SUBAPPLICATION InputOutputTesterButton_AI_Calibrate_3P_OPC_UA (* AI Calibrate 3P Tester (OPC-UA): 8 Analog-Eingaenge mit 3-Punkt-Kalibrierung (Rohwert+kalibrierter Wert+Bargraph+C_MIN/C_MID/C_MAX, fuer Sensoren mit Mittelstellung) + 12 unveraenderte digitale Ausgaenge *)
  (* Standard: 61499-2; Description: Copyright (c) 2026 Meisterschulen am Ostbahnhof This program and the accompanying materials are made available under the terms of the Eclipse Public License 2.0 which is available at https://www.eclipse.org/legal/epl-2.0/ SPDX-License-Identifier: EPL-2.0 *)
  (* Version 1.0, 2026-09-11, Franz Höpfinger, Meisterschulen am Ostbahnhof, 3-Punkt-Pendant zu InputOutputTesterButton_AI_Calibrate_OPC_UA - logiBUS_AI_Calibrate_3P_IDA_OPC statt logiBUS_AI_Calibrate_IDA_OPC (C_MIN/C_MID/C_MAX statt CO/CS) *)
  (* Version 1.1, 2026-09-20, Franz Höpfinger, Meisterschulen am Ostbahnhof, Rohwert-Anzeige an den 3 Kalibrierpunkten (Min/Mid/Max-Raw) fuer alle 8 Kanaele ergaenzt, siehe logiBUS_AI_Calibrate_3P_IDA_OPC v1.8. Neue Parameter stObjMinRaw/stObjMidRaw/stObjMaxRaw + ID_MIN/MID/MAX_RAW_WRITE pro Kanal, neue VT-Objekte NumberVariable_AIC_I0N_MINRAW/_MIDRAW/_MAXRAW_N (DefaultPool_AIC_3P_Numeric, IDs 21040-21063) + OPC-UA-Adressen AIC_I0N_MIN/MID/MAX_RAW_WRITE (SubStrings). *)
  PACKAGE Meins::InputOutputTester::Button_AI_Calibrate_3P_OPC_UA;
  IMPORT Meins::InputOutputTester::Button_AI_Calibrate_3P_OPC_UA::SubStrings::AIC_I1_RAW_WRITE;
  IMPORT Meins::InputOutputTester::Button_AI_Calibrate_3P_OPC_UA::SubStrings::AIC_I1_CAL_WRITE;
  IMPORT Meins::InputOutputTester::Button_AI_Calibrate_3P_OPC_UA::SubStrings::AIC_I2_RAW_WRITE;
  IMPORT Meins::InputOutputTester::Button_AI_Calibrate_3P_OPC_UA::SubStrings::AIC_I2_CAL_WRITE;
  IMPORT Meins::InputOutputTester::Button_AI_Calibrate_3P_OPC_UA::SubStrings::AIC_I3_RAW_WRITE;
  IMPORT Meins::InputOutputTester::Button_AI_Calibrate_3P_OPC_UA::SubStrings::AIC_I3_CAL_WRITE;
  IMPORT Meins::InputOutputTester::Button_AI_Calibrate_3P_OPC_UA::SubStrings::AIC_I4_RAW_WRITE;
  IMPORT Meins::InputOutputTester::Button_AI_Calibrate_3P_OPC_UA::SubStrings::AIC_I4_CAL_WRITE;
  IMPORT Meins::InputOutputTester::Button_AI_Calibrate_3P_OPC_UA::SubStrings::AIC_I5_RAW_WRITE;
  IMPORT Meins::InputOutputTester::Button_AI_Calibrate_3P_OPC_UA::SubStrings::AIC_I5_CAL_WRITE;
  IMPORT Meins::InputOutputTester::Button_AI_Calibrate_3P_OPC_UA::SubStrings::AIC_I6_RAW_WRITE;
  IMPORT Meins::InputOutputTester::Button_AI_Calibrate_3P_OPC_UA::SubStrings::AIC_I6_CAL_WRITE;
  IMPORT Meins::InputOutputTester::Button_AI_Calibrate_3P_OPC_UA::SubStrings::AIC_I7_RAW_WRITE;
  IMPORT Meins::InputOutputTester::Button_AI_Calibrate_3P_OPC_UA::SubStrings::AIC_I7_CAL_WRITE;
  IMPORT Meins::InputOutputTester::Button_AI_Calibrate_3P_OPC_UA::SubStrings::AIC_I8_RAW_WRITE;
  IMPORT Meins::InputOutputTester::Button_AI_Calibrate_3P_OPC_UA::SubStrings::AIC_I8_CAL_WRITE;
  IMPORT Meins::InputOutputTester::Button_AI_Calibrate_3P_OPC_UA::SubStrings::AIC_I1_MIN_METHOD;
  IMPORT Meins::InputOutputTester::Button_AI_Calibrate_3P_OPC_UA::SubStrings::AIC_I1_MID_METHOD;
  IMPORT Meins::InputOutputTester::Button_AI_Calibrate_3P_OPC_UA::SubStrings::AIC_I1_MAX_METHOD;
  IMPORT Meins::InputOutputTester::Button_AI_Calibrate_3P_OPC_UA::SubStrings::AIC_I2_MIN_METHOD;
  IMPORT Meins::InputOutputTester::Button_AI_Calibrate_3P_OPC_UA::SubStrings::AIC_I2_MID_METHOD;
  IMPORT Meins::InputOutputTester::Button_AI_Calibrate_3P_OPC_UA::SubStrings::AIC_I2_MAX_METHOD;
  IMPORT Meins::InputOutputTester::Button_AI_Calibrate_3P_OPC_UA::SubStrings::AIC_I3_MIN_METHOD;
  IMPORT Meins::InputOutputTester::Button_AI_Calibrate_3P_OPC_UA::SubStrings::AIC_I3_MID_METHOD;
  IMPORT Meins::InputOutputTester::Button_AI_Calibrate_3P_OPC_UA::SubStrings::AIC_I3_MAX_METHOD;
  IMPORT Meins::InputOutputTester::Button_AI_Calibrate_3P_OPC_UA::SubStrings::AIC_I4_MIN_METHOD;
  IMPORT Meins::InputOutputTester::Button_AI_Calibrate_3P_OPC_UA::SubStrings::AIC_I4_MID_METHOD;
  IMPORT Meins::InputOutputTester::Button_AI_Calibrate_3P_OPC_UA::SubStrings::AIC_I4_MAX_METHOD;
  IMPORT Meins::InputOutputTester::Button_AI_Calibrate_3P_OPC_UA::SubStrings::AIC_I5_MIN_METHOD;
  IMPORT Meins::InputOutputTester::Button_AI_Calibrate_3P_OPC_UA::SubStrings::AIC_I5_MID_METHOD;
  IMPORT Meins::InputOutputTester::Button_AI_Calibrate_3P_OPC_UA::SubStrings::AIC_I5_MAX_METHOD;
  IMPORT Meins::InputOutputTester::Button_AI_Calibrate_3P_OPC_UA::SubStrings::AIC_I6_MIN_METHOD;
  IMPORT Meins::InputOutputTester::Button_AI_Calibrate_3P_OPC_UA::SubStrings::AIC_I6_MID_METHOD;
  IMPORT Meins::InputOutputTester::Button_AI_Calibrate_3P_OPC_UA::SubStrings::AIC_I6_MAX_METHOD;
  IMPORT Meins::InputOutputTester::Button_AI_Calibrate_3P_OPC_UA::SubStrings::AIC_I7_MIN_METHOD;
  IMPORT Meins::InputOutputTester::Button_AI_Calibrate_3P_OPC_UA::SubStrings::AIC_I7_MID_METHOD;
  IMPORT Meins::InputOutputTester::Button_AI_Calibrate_3P_OPC_UA::SubStrings::AIC_I7_MAX_METHOD;
  IMPORT Meins::InputOutputTester::Button_AI_Calibrate_3P_OPC_UA::SubStrings::AIC_I8_MIN_METHOD;
  IMPORT Meins::InputOutputTester::Button_AI_Calibrate_3P_OPC_UA::SubStrings::AIC_I8_MID_METHOD;
  IMPORT Meins::InputOutputTester::Button_AI_Calibrate_3P_OPC_UA::SubStrings::AIC_I8_MAX_METHOD;
  IMPORT Meins::InputOutputTester::Button_AI_Calibrate_3P_OPC_UA::SubStrings::Q01_READ;
  IMPORT Meins::InputOutputTester::Button_AI_Calibrate_3P_OPC_UA::SubStrings::Q01_WRITE;
  IMPORT Meins::InputOutputTester::Button_AI_Calibrate_3P_OPC_UA::SubStrings::Q02_READ;
  IMPORT Meins::InputOutputTester::Button_AI_Calibrate_3P_OPC_UA::SubStrings::Q02_WRITE;
  IMPORT Meins::InputOutputTester::Button_AI_Calibrate_3P_OPC_UA::SubStrings::Q03_READ;
  IMPORT Meins::InputOutputTester::Button_AI_Calibrate_3P_OPC_UA::SubStrings::Q03_WRITE;
  IMPORT Meins::InputOutputTester::Button_AI_Calibrate_3P_OPC_UA::SubStrings::Q04_READ;
  IMPORT Meins::InputOutputTester::Button_AI_Calibrate_3P_OPC_UA::SubStrings::Q04_WRITE;
  IMPORT Meins::InputOutputTester::Button_AI_Calibrate_3P_OPC_UA::SubStrings::Q05_READ;
  IMPORT Meins::InputOutputTester::Button_AI_Calibrate_3P_OPC_UA::SubStrings::Q05_WRITE;
  IMPORT Meins::InputOutputTester::Button_AI_Calibrate_3P_OPC_UA::SubStrings::Q06_READ;
  IMPORT Meins::InputOutputTester::Button_AI_Calibrate_3P_OPC_UA::SubStrings::Q06_WRITE;
  IMPORT Meins::InputOutputTester::Button_AI_Calibrate_3P_OPC_UA::SubStrings::Q07_READ;
  IMPORT Meins::InputOutputTester::Button_AI_Calibrate_3P_OPC_UA::SubStrings::Q07_WRITE;
  IMPORT Meins::InputOutputTester::Button_AI_Calibrate_3P_OPC_UA::SubStrings::Q08_READ;
  IMPORT Meins::InputOutputTester::Button_AI_Calibrate_3P_OPC_UA::SubStrings::Q08_WRITE;
  IMPORT Meins::InputOutputTester::Button_AI_Calibrate_3P_OPC_UA::SubStrings::Q09_READ;
  IMPORT Meins::InputOutputTester::Button_AI_Calibrate_3P_OPC_UA::SubStrings::Q09_WRITE;
  IMPORT Meins::InputOutputTester::Button_AI_Calibrate_3P_OPC_UA::SubStrings::Q10_READ;
  IMPORT Meins::InputOutputTester::Button_AI_Calibrate_3P_OPC_UA::SubStrings::Q10_WRITE;
  IMPORT Meins::InputOutputTester::Button_AI_Calibrate_3P_OPC_UA::SubStrings::Q11_READ;
  IMPORT Meins::InputOutputTester::Button_AI_Calibrate_3P_OPC_UA::SubStrings::Q11_WRITE;
  IMPORT Meins::InputOutputTester::Button_AI_Calibrate_3P_OPC_UA::SubStrings::Q12_READ;
  IMPORT Meins::InputOutputTester::Button_AI_Calibrate_3P_OPC_UA::SubStrings::Q12_WRITE;
  IMPORT Meins::InputOutputTester::Button_AI_Calibrate_3P_OPC_UA::SubStrings::Tick_WRITE;
  IMPORT Uebungen::const::UT::AIC::DefaultPool_AIC_2P::NumberVariable_AIC_RAW_I01;
  IMPORT Uebungen::const::UT::AIC::DefaultPool_AIC_2P::NumberVariable_AIC_RAW_I02;
  IMPORT Uebungen::const::UT::AIC::DefaultPool_AIC_2P::NumberVariable_AIC_RAW_I03;
  IMPORT Uebungen::const::UT::AIC::DefaultPool_AIC_2P::NumberVariable_AIC_RAW_I04;
  IMPORT Uebungen::const::UT::AIC::DefaultPool_AIC_2P::NumberVariable_AIC_RAW_I05;
  IMPORT Uebungen::const::UT::AIC::DefaultPool_AIC_2P::NumberVariable_AIC_RAW_I06;
  IMPORT Uebungen::const::UT::AIC::DefaultPool_AIC_2P::NumberVariable_AIC_RAW_I07;
  IMPORT Uebungen::const::UT::AIC::DefaultPool_AIC_2P::NumberVariable_AIC_RAW_I08;
  IMPORT Uebungen::const::UT::AIC::DefaultPool_AIC_3P_Numeric::NumberVariable_AIC_CAL_I01_N;
  IMPORT Uebungen::const::UT::AIC::DefaultPool_AIC_3P_Numeric::NumberVariable_AIC_CAL_I02_N;
  IMPORT Uebungen::const::UT::AIC::DefaultPool_AIC_3P_Numeric::NumberVariable_AIC_CAL_I03_N;
  IMPORT Uebungen::const::UT::AIC::DefaultPool_AIC_3P_Numeric::NumberVariable_AIC_CAL_I04_N;
  IMPORT Uebungen::const::UT::AIC::DefaultPool_AIC_3P_Numeric::NumberVariable_AIC_CAL_I05_N;
  IMPORT Uebungen::const::UT::AIC::DefaultPool_AIC_3P_Numeric::NumberVariable_AIC_CAL_I06_N;
  IMPORT Uebungen::const::UT::AIC::DefaultPool_AIC_3P_Numeric::NumberVariable_AIC_CAL_I07_N;
  IMPORT Uebungen::const::UT::AIC::DefaultPool_AIC_3P_Numeric::NumberVariable_AIC_CAL_I08_N;
  IMPORT Uebungen::const::UT::AIC::DefaultPool_AIC_3P::Button_AIC_I01_CO;
  IMPORT Uebungen::const::UT::AIC::DefaultPool_AIC_3P::Button_AIC_I01_MID;
  IMPORT Uebungen::const::UT::AIC::DefaultPool_AIC_3P::Button_AIC_I01_CS;
  IMPORT Uebungen::const::UT::AIC::DefaultPool_AIC_3P::Button_AIC_I02_CO;
  IMPORT Uebungen::const::UT::AIC::DefaultPool_AIC_3P::Button_AIC_I02_MID;
  IMPORT Uebungen::const::UT::AIC::DefaultPool_AIC_3P::Button_AIC_I02_CS;
  IMPORT Uebungen::const::UT::AIC::DefaultPool_AIC_3P::Button_AIC_I03_CO;
  IMPORT Uebungen::const::UT::AIC::DefaultPool_AIC_3P::Button_AIC_I03_MID;
  IMPORT Uebungen::const::UT::AIC::DefaultPool_AIC_3P::Button_AIC_I03_CS;
  IMPORT Uebungen::const::UT::AIC::DefaultPool_AIC_3P::Button_AIC_I04_CO;
  IMPORT Uebungen::const::UT::AIC::DefaultPool_AIC_3P::Button_AIC_I04_MID;
  IMPORT Uebungen::const::UT::AIC::DefaultPool_AIC_3P::Button_AIC_I04_CS;
  IMPORT Uebungen::const::UT::AIC::DefaultPool_AIC_3P::Button_AIC_I05_CO;
  IMPORT Uebungen::const::UT::AIC::DefaultPool_AIC_3P::Button_AIC_I05_MID;
  IMPORT Uebungen::const::UT::AIC::DefaultPool_AIC_3P::Button_AIC_I05_CS;
  IMPORT Uebungen::const::UT::AIC::DefaultPool_AIC_3P::Button_AIC_I06_CO;
  IMPORT Uebungen::const::UT::AIC::DefaultPool_AIC_3P::Button_AIC_I06_MID;
  IMPORT Uebungen::const::UT::AIC::DefaultPool_AIC_3P::Button_AIC_I06_CS;
  IMPORT Uebungen::const::UT::AIC::DefaultPool_AIC_3P::Button_AIC_I07_CO;
  IMPORT Uebungen::const::UT::AIC::DefaultPool_AIC_3P::Button_AIC_I07_MID;
  IMPORT Uebungen::const::UT::AIC::DefaultPool_AIC_3P::Button_AIC_I07_CS;
  IMPORT Uebungen::const::UT::AIC::DefaultPool_AIC_3P::Button_AIC_I08_CO;
  IMPORT Uebungen::const::UT::AIC::DefaultPool_AIC_3P::Button_AIC_I08_MID;
  IMPORT Uebungen::const::UT::AIC::DefaultPool_AIC_3P::Button_AIC_I08_CS;
  IMPORT Uebungen::const::UT::AIC::DefaultPool_AIC_2P::Button_Q01;
  IMPORT Uebungen::const::UT::AIC::DefaultPool_AIC_2P::Button_Q02;
  IMPORT Uebungen::const::UT::AIC::DefaultPool_AIC_2P::Button_Q03;
  IMPORT Uebungen::const::UT::AIC::DefaultPool_AIC_2P::Button_Q04;
  IMPORT Uebungen::const::UT::AIC::DefaultPool_AIC_2P::Button_Q05;
  IMPORT Uebungen::const::UT::AIC::DefaultPool_AIC_2P::Button_Q06;
  IMPORT Uebungen::const::UT::AIC::DefaultPool_AIC_2P::Button_Q07;
  IMPORT Uebungen::const::UT::AIC::DefaultPool_AIC_2P::Button_Q08;
  IMPORT Uebungen::const::UT::AIC::DefaultPool_AIC_2P::Button_Q09;
  IMPORT Uebungen::const::UT::AIC::DefaultPool_AIC_2P::Button_Q10;
  IMPORT Uebungen::const::UT::AIC::DefaultPool_AIC_2P::Button_Q11;
  IMPORT Uebungen::const::UT::AIC::DefaultPool_AIC_2P::Button_Q12;
  IMPORT Uebungen::const::UT::AIC::DefaultPool_AIC_2P::OutputNumber_Tick;
  IMPORT logiBUS::io::AI::logiBUS_AI::AnalogInput_I1;
  IMPORT logiBUS::io::AI::logiBUS_AI::AnalogInput_I2;
  IMPORT logiBUS::io::AI::logiBUS_AI::AnalogInput_I3;
  IMPORT logiBUS::io::AI::logiBUS_AI::AnalogInput_I4;
  IMPORT logiBUS::io::AI::logiBUS_AI::AnalogInput_I5;
  IMPORT logiBUS::io::AI::logiBUS_AI::AnalogInput_I6;
  IMPORT logiBUS::io::AI::logiBUS_AI::AnalogInput_I7;
  IMPORT logiBUS::io::AI::logiBUS_AI::AnalogInput_I8;
  IMPORT logiBUS::io::DQ::logiBUS_DO::Output_Q1;
  IMPORT logiBUS::io::DQ::logiBUS_DO::Output_Q10;
  IMPORT logiBUS::io::DQ::logiBUS_DO::Output_Q11;
  IMPORT logiBUS::io::DQ::logiBUS_DO::Output_Q12;
  IMPORT logiBUS::io::DQ::logiBUS_DO::Output_Q2;
  IMPORT logiBUS::io::DQ::logiBUS_DO::Output_Q3;
  IMPORT logiBUS::io::DQ::logiBUS_DO::Output_Q4;
  IMPORT logiBUS::io::DQ::logiBUS_DO::Output_Q5;
  IMPORT logiBUS::io::DQ::logiBUS_DO::Output_Q6;
  IMPORT logiBUS::io::DQ::logiBUS_DO::Output_Q7;
  IMPORT logiBUS::io::DQ::logiBUS_DO::Output_Q8;
  IMPORT logiBUS::io::DQ::logiBUS_DO::Output_Q9;
  IMPORT Meins::InputOutputTester::Button_AI_Calibrate_3P_OPC_UA::SubStrings::AIC_I1_MINREF_READ;
  IMPORT Meins::InputOutputTester::Button_AI_Calibrate_3P_OPC_UA::SubStrings::AIC_I1_MINREF_WRITE;
  IMPORT Meins::InputOutputTester::Button_AI_Calibrate_3P_OPC_UA::SubStrings::AIC_I1_MIDREF_READ;
  IMPORT Meins::InputOutputTester::Button_AI_Calibrate_3P_OPC_UA::SubStrings::AIC_I1_MIDREF_WRITE;
  IMPORT Meins::InputOutputTester::Button_AI_Calibrate_3P_OPC_UA::SubStrings::AIC_I1_MAXREF_READ;
  IMPORT Meins::InputOutputTester::Button_AI_Calibrate_3P_OPC_UA::SubStrings::AIC_I1_MAXREF_WRITE;
  IMPORT Meins::InputOutputTester::Button_AI_Calibrate_3P_OPC_UA::SubStrings::AIC_I2_MINREF_READ;
  IMPORT Meins::InputOutputTester::Button_AI_Calibrate_3P_OPC_UA::SubStrings::AIC_I2_MINREF_WRITE;
  IMPORT Meins::InputOutputTester::Button_AI_Calibrate_3P_OPC_UA::SubStrings::AIC_I2_MIDREF_READ;
  IMPORT Meins::InputOutputTester::Button_AI_Calibrate_3P_OPC_UA::SubStrings::AIC_I2_MIDREF_WRITE;
  IMPORT Meins::InputOutputTester::Button_AI_Calibrate_3P_OPC_UA::SubStrings::AIC_I2_MAXREF_READ;
  IMPORT Meins::InputOutputTester::Button_AI_Calibrate_3P_OPC_UA::SubStrings::AIC_I2_MAXREF_WRITE;
  IMPORT Meins::InputOutputTester::Button_AI_Calibrate_3P_OPC_UA::SubStrings::AIC_I3_MINREF_READ;
  IMPORT Meins::InputOutputTester::Button_AI_Calibrate_3P_OPC_UA::SubStrings::AIC_I3_MINREF_WRITE;
  IMPORT Meins::InputOutputTester::Button_AI_Calibrate_3P_OPC_UA::SubStrings::AIC_I3_MIDREF_READ;
  IMPORT Meins::InputOutputTester::Button_AI_Calibrate_3P_OPC_UA::SubStrings::AIC_I3_MIDREF_WRITE;
  IMPORT Meins::InputOutputTester::Button_AI_Calibrate_3P_OPC_UA::SubStrings::AIC_I3_MAXREF_READ;
  IMPORT Meins::InputOutputTester::Button_AI_Calibrate_3P_OPC_UA::SubStrings::AIC_I3_MAXREF_WRITE;
  IMPORT Meins::InputOutputTester::Button_AI_Calibrate_3P_OPC_UA::SubStrings::AIC_I4_MINREF_READ;
  IMPORT Meins::InputOutputTester::Button_AI_Calibrate_3P_OPC_UA::SubStrings::AIC_I4_MINREF_WRITE;
  IMPORT Meins::InputOutputTester::Button_AI_Calibrate_3P_OPC_UA::SubStrings::AIC_I4_MIDREF_READ;
  IMPORT Meins::InputOutputTester::Button_AI_Calibrate_3P_OPC_UA::SubStrings::AIC_I4_MIDREF_WRITE;
  IMPORT Meins::InputOutputTester::Button_AI_Calibrate_3P_OPC_UA::SubStrings::AIC_I4_MAXREF_READ;
  IMPORT Meins::InputOutputTester::Button_AI_Calibrate_3P_OPC_UA::SubStrings::AIC_I4_MAXREF_WRITE;
  IMPORT Meins::InputOutputTester::Button_AI_Calibrate_3P_OPC_UA::SubStrings::AIC_I5_MINREF_READ;
  IMPORT Meins::InputOutputTester::Button_AI_Calibrate_3P_OPC_UA::SubStrings::AIC_I5_MINREF_WRITE;
  IMPORT Meins::InputOutputTester::Button_AI_Calibrate_3P_OPC_UA::SubStrings::AIC_I5_MIDREF_READ;
  IMPORT Meins::InputOutputTester::Button_AI_Calibrate_3P_OPC_UA::SubStrings::AIC_I5_MIDREF_WRITE;
  IMPORT Meins::InputOutputTester::Button_AI_Calibrate_3P_OPC_UA::SubStrings::AIC_I5_MAXREF_READ;
  IMPORT Meins::InputOutputTester::Button_AI_Calibrate_3P_OPC_UA::SubStrings::AIC_I5_MAXREF_WRITE;
  IMPORT Meins::InputOutputTester::Button_AI_Calibrate_3P_OPC_UA::SubStrings::AIC_I6_MINREF_READ;
  IMPORT Meins::InputOutputTester::Button_AI_Calibrate_3P_OPC_UA::SubStrings::AIC_I6_MINREF_WRITE;
  IMPORT Meins::InputOutputTester::Button_AI_Calibrate_3P_OPC_UA::SubStrings::AIC_I6_MIDREF_READ;
  IMPORT Meins::InputOutputTester::Button_AI_Calibrate_3P_OPC_UA::SubStrings::AIC_I6_MIDREF_WRITE;
  IMPORT Meins::InputOutputTester::Button_AI_Calibrate_3P_OPC_UA::SubStrings::AIC_I6_MAXREF_READ;
  IMPORT Meins::InputOutputTester::Button_AI_Calibrate_3P_OPC_UA::SubStrings::AIC_I6_MAXREF_WRITE;
  IMPORT Meins::InputOutputTester::Button_AI_Calibrate_3P_OPC_UA::SubStrings::AIC_I7_MINREF_READ;
  IMPORT Meins::InputOutputTester::Button_AI_Calibrate_3P_OPC_UA::SubStrings::AIC_I7_MINREF_WRITE;
  IMPORT Meins::InputOutputTester::Button_AI_Calibrate_3P_OPC_UA::SubStrings::AIC_I7_MIDREF_READ;
  IMPORT Meins::InputOutputTester::Button_AI_Calibrate_3P_OPC_UA::SubStrings::AIC_I7_MIDREF_WRITE;
  IMPORT Meins::InputOutputTester::Button_AI_Calibrate_3P_OPC_UA::SubStrings::AIC_I7_MAXREF_READ;
  IMPORT Meins::InputOutputTester::Button_AI_Calibrate_3P_OPC_UA::SubStrings::AIC_I7_MAXREF_WRITE;
  IMPORT Meins::InputOutputTester::Button_AI_Calibrate_3P_OPC_UA::SubStrings::AIC_I8_MINREF_READ;
  IMPORT Meins::InputOutputTester::Button_AI_Calibrate_3P_OPC_UA::SubStrings::AIC_I8_MINREF_WRITE;
  IMPORT Meins::InputOutputTester::Button_AI_Calibrate_3P_OPC_UA::SubStrings::AIC_I8_MIDREF_READ;
  IMPORT Meins::InputOutputTester::Button_AI_Calibrate_3P_OPC_UA::SubStrings::AIC_I8_MIDREF_WRITE;
  IMPORT Meins::InputOutputTester::Button_AI_Calibrate_3P_OPC_UA::SubStrings::AIC_I8_MAXREF_READ;
  IMPORT Meins::InputOutputTester::Button_AI_Calibrate_3P_OPC_UA::SubStrings::AIC_I8_MAXREF_WRITE;
  IMPORT Meins::InputOutputTester::Button_AI_Calibrate_3P_OPC_UA::SubStrings::AIC_I1_MIN_RAW_WRITE;
  IMPORT Meins::InputOutputTester::Button_AI_Calibrate_3P_OPC_UA::SubStrings::AIC_I1_MID_RAW_WRITE;
  IMPORT Meins::InputOutputTester::Button_AI_Calibrate_3P_OPC_UA::SubStrings::AIC_I1_MAX_RAW_WRITE;
  IMPORT Meins::InputOutputTester::Button_AI_Calibrate_3P_OPC_UA::SubStrings::AIC_I2_MIN_RAW_WRITE;
  IMPORT Meins::InputOutputTester::Button_AI_Calibrate_3P_OPC_UA::SubStrings::AIC_I2_MID_RAW_WRITE;
  IMPORT Meins::InputOutputTester::Button_AI_Calibrate_3P_OPC_UA::SubStrings::AIC_I2_MAX_RAW_WRITE;
  IMPORT Meins::InputOutputTester::Button_AI_Calibrate_3P_OPC_UA::SubStrings::AIC_I3_MIN_RAW_WRITE;
  IMPORT Meins::InputOutputTester::Button_AI_Calibrate_3P_OPC_UA::SubStrings::AIC_I3_MID_RAW_WRITE;
  IMPORT Meins::InputOutputTester::Button_AI_Calibrate_3P_OPC_UA::SubStrings::AIC_I3_MAX_RAW_WRITE;
  IMPORT Meins::InputOutputTester::Button_AI_Calibrate_3P_OPC_UA::SubStrings::AIC_I4_MIN_RAW_WRITE;
  IMPORT Meins::InputOutputTester::Button_AI_Calibrate_3P_OPC_UA::SubStrings::AIC_I4_MID_RAW_WRITE;
  IMPORT Meins::InputOutputTester::Button_AI_Calibrate_3P_OPC_UA::SubStrings::AIC_I4_MAX_RAW_WRITE;
  IMPORT Meins::InputOutputTester::Button_AI_Calibrate_3P_OPC_UA::SubStrings::AIC_I5_MIN_RAW_WRITE;
  IMPORT Meins::InputOutputTester::Button_AI_Calibrate_3P_OPC_UA::SubStrings::AIC_I5_MID_RAW_WRITE;
  IMPORT Meins::InputOutputTester::Button_AI_Calibrate_3P_OPC_UA::SubStrings::AIC_I5_MAX_RAW_WRITE;
  IMPORT Meins::InputOutputTester::Button_AI_Calibrate_3P_OPC_UA::SubStrings::AIC_I6_MIN_RAW_WRITE;
  IMPORT Meins::InputOutputTester::Button_AI_Calibrate_3P_OPC_UA::SubStrings::AIC_I6_MID_RAW_WRITE;
  IMPORT Meins::InputOutputTester::Button_AI_Calibrate_3P_OPC_UA::SubStrings::AIC_I6_MAX_RAW_WRITE;
  IMPORT Meins::InputOutputTester::Button_AI_Calibrate_3P_OPC_UA::SubStrings::AIC_I7_MIN_RAW_WRITE;
  IMPORT Meins::InputOutputTester::Button_AI_Calibrate_3P_OPC_UA::SubStrings::AIC_I7_MID_RAW_WRITE;
  IMPORT Meins::InputOutputTester::Button_AI_Calibrate_3P_OPC_UA::SubStrings::AIC_I7_MAX_RAW_WRITE;
  IMPORT Meins::InputOutputTester::Button_AI_Calibrate_3P_OPC_UA::SubStrings::AIC_I8_MIN_RAW_WRITE;
  IMPORT Meins::InputOutputTester::Button_AI_Calibrate_3P_OPC_UA::SubStrings::AIC_I8_MID_RAW_WRITE;
  IMPORT Meins::InputOutputTester::Button_AI_Calibrate_3P_OPC_UA::SubStrings::AIC_I8_MAX_RAW_WRITE;
  IMPORT Uebungen::const::UT::AIC::DefaultPool_AIC_3P_Numeric::NumberVariable_AIC_I01_ZERO_N;
  IMPORT Uebungen::const::UT::AIC::DefaultPool_AIC_3P_Numeric::NumberVariable_AIC_I01_MID_N;
  IMPORT Uebungen::const::UT::AIC::DefaultPool_AIC_3P_Numeric::NumberVariable_AIC_I01_SPAN_N;
  IMPORT Uebungen::const::UT::AIC::DefaultPool_AIC_3P_Numeric::NumberVariable_AIC_I02_ZERO_N;
  IMPORT Uebungen::const::UT::AIC::DefaultPool_AIC_3P_Numeric::NumberVariable_AIC_I02_MID_N;
  IMPORT Uebungen::const::UT::AIC::DefaultPool_AIC_3P_Numeric::NumberVariable_AIC_I02_SPAN_N;
  IMPORT Uebungen::const::UT::AIC::DefaultPool_AIC_3P_Numeric::NumberVariable_AIC_I03_ZERO_N;
  IMPORT Uebungen::const::UT::AIC::DefaultPool_AIC_3P_Numeric::NumberVariable_AIC_I03_MID_N;
  IMPORT Uebungen::const::UT::AIC::DefaultPool_AIC_3P_Numeric::NumberVariable_AIC_I03_SPAN_N;
  IMPORT Uebungen::const::UT::AIC::DefaultPool_AIC_3P_Numeric::NumberVariable_AIC_I04_ZERO_N;
  IMPORT Uebungen::const::UT::AIC::DefaultPool_AIC_3P_Numeric::NumberVariable_AIC_I04_MID_N;
  IMPORT Uebungen::const::UT::AIC::DefaultPool_AIC_3P_Numeric::NumberVariable_AIC_I04_SPAN_N;
  IMPORT Uebungen::const::UT::AIC::DefaultPool_AIC_3P_Numeric::NumberVariable_AIC_I05_ZERO_N;
  IMPORT Uebungen::const::UT::AIC::DefaultPool_AIC_3P_Numeric::NumberVariable_AIC_I05_MID_N;
  IMPORT Uebungen::const::UT::AIC::DefaultPool_AIC_3P_Numeric::NumberVariable_AIC_I05_SPAN_N;
  IMPORT Uebungen::const::UT::AIC::DefaultPool_AIC_3P_Numeric::NumberVariable_AIC_I06_ZERO_N;
  IMPORT Uebungen::const::UT::AIC::DefaultPool_AIC_3P_Numeric::NumberVariable_AIC_I06_MID_N;
  IMPORT Uebungen::const::UT::AIC::DefaultPool_AIC_3P_Numeric::NumberVariable_AIC_I06_SPAN_N;
  IMPORT Uebungen::const::UT::AIC::DefaultPool_AIC_3P_Numeric::NumberVariable_AIC_I07_ZERO_N;
  IMPORT Uebungen::const::UT::AIC::DefaultPool_AIC_3P_Numeric::NumberVariable_AIC_I07_MID_N;
  IMPORT Uebungen::const::UT::AIC::DefaultPool_AIC_3P_Numeric::NumberVariable_AIC_I07_SPAN_N;
  IMPORT Uebungen::const::UT::AIC::DefaultPool_AIC_3P_Numeric::NumberVariable_AIC_I08_ZERO_N;
  IMPORT Uebungen::const::UT::AIC::DefaultPool_AIC_3P_Numeric::NumberVariable_AIC_I08_MID_N;
  IMPORT Uebungen::const::UT::AIC::DefaultPool_AIC_3P_Numeric::NumberVariable_AIC_I08_SPAN_N;
  IMPORT Uebungen::const::UT::AIC::DefaultPool_AIC_3P_Numeric::NumberVariable_AIC_I01_MINRAW_N;
  IMPORT Uebungen::const::UT::AIC::DefaultPool_AIC_3P_Numeric::NumberVariable_AIC_I01_MIDRAW_N;
  IMPORT Uebungen::const::UT::AIC::DefaultPool_AIC_3P_Numeric::NumberVariable_AIC_I01_MAXRAW_N;
  IMPORT Uebungen::const::UT::AIC::DefaultPool_AIC_3P_Numeric::NumberVariable_AIC_I02_MINRAW_N;
  IMPORT Uebungen::const::UT::AIC::DefaultPool_AIC_3P_Numeric::NumberVariable_AIC_I02_MIDRAW_N;
  IMPORT Uebungen::const::UT::AIC::DefaultPool_AIC_3P_Numeric::NumberVariable_AIC_I02_MAXRAW_N;
  IMPORT Uebungen::const::UT::AIC::DefaultPool_AIC_3P_Numeric::NumberVariable_AIC_I03_MINRAW_N;
  IMPORT Uebungen::const::UT::AIC::DefaultPool_AIC_3P_Numeric::NumberVariable_AIC_I03_MIDRAW_N;
  IMPORT Uebungen::const::UT::AIC::DefaultPool_AIC_3P_Numeric::NumberVariable_AIC_I03_MAXRAW_N;
  IMPORT Uebungen::const::UT::AIC::DefaultPool_AIC_3P_Numeric::NumberVariable_AIC_I04_MINRAW_N;
  IMPORT Uebungen::const::UT::AIC::DefaultPool_AIC_3P_Numeric::NumberVariable_AIC_I04_MIDRAW_N;
  IMPORT Uebungen::const::UT::AIC::DefaultPool_AIC_3P_Numeric::NumberVariable_AIC_I04_MAXRAW_N;
  IMPORT Uebungen::const::UT::AIC::DefaultPool_AIC_3P_Numeric::NumberVariable_AIC_I05_MINRAW_N;
  IMPORT Uebungen::const::UT::AIC::DefaultPool_AIC_3P_Numeric::NumberVariable_AIC_I05_MIDRAW_N;
  IMPORT Uebungen::const::UT::AIC::DefaultPool_AIC_3P_Numeric::NumberVariable_AIC_I05_MAXRAW_N;
  IMPORT Uebungen::const::UT::AIC::DefaultPool_AIC_3P_Numeric::NumberVariable_AIC_I06_MINRAW_N;
  IMPORT Uebungen::const::UT::AIC::DefaultPool_AIC_3P_Numeric::NumberVariable_AIC_I06_MIDRAW_N;
  IMPORT Uebungen::const::UT::AIC::DefaultPool_AIC_3P_Numeric::NumberVariable_AIC_I06_MAXRAW_N;
  IMPORT Uebungen::const::UT::AIC::DefaultPool_AIC_3P_Numeric::NumberVariable_AIC_I07_MINRAW_N;
  IMPORT Uebungen::const::UT::AIC::DefaultPool_AIC_3P_Numeric::NumberVariable_AIC_I07_MIDRAW_N;
  IMPORT Uebungen::const::UT::AIC::DefaultPool_AIC_3P_Numeric::NumberVariable_AIC_I07_MAXRAW_N;
  IMPORT Uebungen::const::UT::AIC::DefaultPool_AIC_3P_Numeric::NumberVariable_AIC_I08_MINRAW_N;
  IMPORT Uebungen::const::UT::AIC::DefaultPool_AIC_3P_Numeric::NumberVariable_AIC_I08_MIDRAW_N;
  IMPORT Uebungen::const::UT::AIC::DefaultPool_AIC_3P_Numeric::NumberVariable_AIC_I08_MAXRAW_N;
  SUBAPPS
    AnalogChannel_I1 : MyLib::sys::logiBUS_AI_Calibrate_3P_IDA_OPC(u16ObjId_RAWVAR := NumberVariable_AIC_RAW_I01, stObjCal := NumberVariable_AIC_CAL_I01_N, u16ObjId_C_MIN := Button_AIC_I01_CO, u16ObjId_C_MID := Button_AIC_I01_MID, u16ObjId_C_MAX := Button_AIC_I01_CS, Input := AnalogInput_I1, sSection := 'AI_Calibrate_3P_I1', ID_RAW_WRITE := AIC_I1_RAW_WRITE, ID_CAL_WRITE := AIC_I1_CAL_WRITE, ID_MIN_METHOD := AIC_I1_MIN_METHOD, ID_MID_TRIGGER_METHOD := AIC_I1_MID_METHOD, ID_MAX_METHOD := AIC_I1_MAX_METHOD, stObjMinRef := NumberVariable_AIC_I01_ZERO_N, stObjMidRef := NumberVariable_AIC_I01_MID_N, stObjMaxRef := NumberVariable_AIC_I01_SPAN_N, ID_MINREF_READ := AIC_I1_MINREF_READ, ID_MINREF_WRITE := AIC_I1_MINREF_WRITE, ID_MIDREF_READ := AIC_I1_MIDREF_READ, ID_MIDREF_WRITE := AIC_I1_MIDREF_WRITE, ID_MAXREF_READ := AIC_I1_MAXREF_READ, ID_MAXREF_WRITE := AIC_I1_MAXREF_WRITE, stObjMinRaw := NumberVariable_AIC_I01_MINRAW_N, stObjMidRaw := NumberVariable_AIC_I01_MIDRAW_N, stObjMaxRaw := NumberVariable_AIC_I01_MAXRAW_N, ID_MIN_RAW_WRITE := AIC_I1_MIN_RAW_WRITE, ID_MID_RAW_WRITE := AIC_I1_MID_RAW_WRITE, ID_MAX_RAW_WRITE := AIC_I1_MAX_RAW_WRITE);
    AnalogChannel_I2 : MyLib::sys::logiBUS_AI_Calibrate_3P_IDA_OPC(u16ObjId_RAWVAR := NumberVariable_AIC_RAW_I02, stObjCal := NumberVariable_AIC_CAL_I02_N, u16ObjId_C_MIN := Button_AIC_I02_CO, u16ObjId_C_MID := Button_AIC_I02_MID, u16ObjId_C_MAX := Button_AIC_I02_CS, Input := AnalogInput_I2, sSection := 'AI_Calibrate_3P_I2', ID_RAW_WRITE := AIC_I2_RAW_WRITE, ID_CAL_WRITE := AIC_I2_CAL_WRITE, ID_MIN_METHOD := AIC_I2_MIN_METHOD, ID_MID_TRIGGER_METHOD := AIC_I2_MID_METHOD, ID_MAX_METHOD := AIC_I2_MAX_METHOD, stObjMinRef := NumberVariable_AIC_I02_ZERO_N, stObjMidRef := NumberVariable_AIC_I02_MID_N, stObjMaxRef := NumberVariable_AIC_I02_SPAN_N, ID_MINREF_READ := AIC_I2_MINREF_READ, ID_MINREF_WRITE := AIC_I2_MINREF_WRITE, ID_MIDREF_READ := AIC_I2_MIDREF_READ, ID_MIDREF_WRITE := AIC_I2_MIDREF_WRITE, ID_MAXREF_READ := AIC_I2_MAXREF_READ, ID_MAXREF_WRITE := AIC_I2_MAXREF_WRITE, stObjMinRaw := NumberVariable_AIC_I02_MINRAW_N, stObjMidRaw := NumberVariable_AIC_I02_MIDRAW_N, stObjMaxRaw := NumberVariable_AIC_I02_MAXRAW_N, ID_MIN_RAW_WRITE := AIC_I2_MIN_RAW_WRITE, ID_MID_RAW_WRITE := AIC_I2_MID_RAW_WRITE, ID_MAX_RAW_WRITE := AIC_I2_MAX_RAW_WRITE);
    AnalogChannel_I3 : MyLib::sys::logiBUS_AI_Calibrate_3P_IDA_OPC(u16ObjId_RAWVAR := NumberVariable_AIC_RAW_I03, stObjCal := NumberVariable_AIC_CAL_I03_N, u16ObjId_C_MIN := Button_AIC_I03_CO, u16ObjId_C_MID := Button_AIC_I03_MID, u16ObjId_C_MAX := Button_AIC_I03_CS, Input := AnalogInput_I3, sSection := 'AI_Calibrate_3P_I3', ID_RAW_WRITE := AIC_I3_RAW_WRITE, ID_CAL_WRITE := AIC_I3_CAL_WRITE, ID_MIN_METHOD := AIC_I3_MIN_METHOD, ID_MID_TRIGGER_METHOD := AIC_I3_MID_METHOD, ID_MAX_METHOD := AIC_I3_MAX_METHOD, stObjMinRef := NumberVariable_AIC_I03_ZERO_N, stObjMidRef := NumberVariable_AIC_I03_MID_N, stObjMaxRef := NumberVariable_AIC_I03_SPAN_N, ID_MINREF_READ := AIC_I3_MINREF_READ, ID_MINREF_WRITE := AIC_I3_MINREF_WRITE, ID_MIDREF_READ := AIC_I3_MIDREF_READ, ID_MIDREF_WRITE := AIC_I3_MIDREF_WRITE, ID_MAXREF_READ := AIC_I3_MAXREF_READ, ID_MAXREF_WRITE := AIC_I3_MAXREF_WRITE, stObjMinRaw := NumberVariable_AIC_I03_MINRAW_N, stObjMidRaw := NumberVariable_AIC_I03_MIDRAW_N, stObjMaxRaw := NumberVariable_AIC_I03_MAXRAW_N, ID_MIN_RAW_WRITE := AIC_I3_MIN_RAW_WRITE, ID_MID_RAW_WRITE := AIC_I3_MID_RAW_WRITE, ID_MAX_RAW_WRITE := AIC_I3_MAX_RAW_WRITE);
    AnalogChannel_I4 : MyLib::sys::logiBUS_AI_Calibrate_3P_IDA_OPC(u16ObjId_RAWVAR := NumberVariable_AIC_RAW_I04, stObjCal := NumberVariable_AIC_CAL_I04_N, u16ObjId_C_MIN := Button_AIC_I04_CO, u16ObjId_C_MID := Button_AIC_I04_MID, u16ObjId_C_MAX := Button_AIC_I04_CS, Input := AnalogInput_I4, sSection := 'AI_Calibrate_3P_I4', ID_RAW_WRITE := AIC_I4_RAW_WRITE, ID_CAL_WRITE := AIC_I4_CAL_WRITE, ID_MIN_METHOD := AIC_I4_MIN_METHOD, ID_MID_TRIGGER_METHOD := AIC_I4_MID_METHOD, ID_MAX_METHOD := AIC_I4_MAX_METHOD, stObjMinRef := NumberVariable_AIC_I04_ZERO_N, stObjMidRef := NumberVariable_AIC_I04_MID_N, stObjMaxRef := NumberVariable_AIC_I04_SPAN_N, ID_MINREF_READ := AIC_I4_MINREF_READ, ID_MINREF_WRITE := AIC_I4_MINREF_WRITE, ID_MIDREF_READ := AIC_I4_MIDREF_READ, ID_MIDREF_WRITE := AIC_I4_MIDREF_WRITE, ID_MAXREF_READ := AIC_I4_MAXREF_READ, ID_MAXREF_WRITE := AIC_I4_MAXREF_WRITE, stObjMinRaw := NumberVariable_AIC_I04_MINRAW_N, stObjMidRaw := NumberVariable_AIC_I04_MIDRAW_N, stObjMaxRaw := NumberVariable_AIC_I04_MAXRAW_N, ID_MIN_RAW_WRITE := AIC_I4_MIN_RAW_WRITE, ID_MID_RAW_WRITE := AIC_I4_MID_RAW_WRITE, ID_MAX_RAW_WRITE := AIC_I4_MAX_RAW_WRITE);
    AnalogChannel_I5 : MyLib::sys::logiBUS_AI_Calibrate_3P_IDA_OPC(u16ObjId_RAWVAR := NumberVariable_AIC_RAW_I05, stObjCal := NumberVariable_AIC_CAL_I05_N, u16ObjId_C_MIN := Button_AIC_I05_CO, u16ObjId_C_MID := Button_AIC_I05_MID, u16ObjId_C_MAX := Button_AIC_I05_CS, Input := AnalogInput_I5, sSection := 'AI_Calibrate_3P_I5', ID_RAW_WRITE := AIC_I5_RAW_WRITE, ID_CAL_WRITE := AIC_I5_CAL_WRITE, ID_MIN_METHOD := AIC_I5_MIN_METHOD, ID_MID_TRIGGER_METHOD := AIC_I5_MID_METHOD, ID_MAX_METHOD := AIC_I5_MAX_METHOD, stObjMinRef := NumberVariable_AIC_I05_ZERO_N, stObjMidRef := NumberVariable_AIC_I05_MID_N, stObjMaxRef := NumberVariable_AIC_I05_SPAN_N, ID_MINREF_READ := AIC_I5_MINREF_READ, ID_MINREF_WRITE := AIC_I5_MINREF_WRITE, ID_MIDREF_READ := AIC_I5_MIDREF_READ, ID_MIDREF_WRITE := AIC_I5_MIDREF_WRITE, ID_MAXREF_READ := AIC_I5_MAXREF_READ, ID_MAXREF_WRITE := AIC_I5_MAXREF_WRITE, stObjMinRaw := NumberVariable_AIC_I05_MINRAW_N, stObjMidRaw := NumberVariable_AIC_I05_MIDRAW_N, stObjMaxRaw := NumberVariable_AIC_I05_MAXRAW_N, ID_MIN_RAW_WRITE := AIC_I5_MIN_RAW_WRITE, ID_MID_RAW_WRITE := AIC_I5_MID_RAW_WRITE, ID_MAX_RAW_WRITE := AIC_I5_MAX_RAW_WRITE);
    AnalogChannel_I6 : MyLib::sys::logiBUS_AI_Calibrate_3P_IDA_OPC(u16ObjId_RAWVAR := NumberVariable_AIC_RAW_I06, stObjCal := NumberVariable_AIC_CAL_I06_N, u16ObjId_C_MIN := Button_AIC_I06_CO, u16ObjId_C_MID := Button_AIC_I06_MID, u16ObjId_C_MAX := Button_AIC_I06_CS, Input := AnalogInput_I6, sSection := 'AI_Calibrate_3P_I6', ID_RAW_WRITE := AIC_I6_RAW_WRITE, ID_CAL_WRITE := AIC_I6_CAL_WRITE, ID_MIN_METHOD := AIC_I6_MIN_METHOD, ID_MID_TRIGGER_METHOD := AIC_I6_MID_METHOD, ID_MAX_METHOD := AIC_I6_MAX_METHOD, stObjMinRef := NumberVariable_AIC_I06_ZERO_N, stObjMidRef := NumberVariable_AIC_I06_MID_N, stObjMaxRef := NumberVariable_AIC_I06_SPAN_N, ID_MINREF_READ := AIC_I6_MINREF_READ, ID_MINREF_WRITE := AIC_I6_MINREF_WRITE, ID_MIDREF_READ := AIC_I6_MIDREF_READ, ID_MIDREF_WRITE := AIC_I6_MIDREF_WRITE, ID_MAXREF_READ := AIC_I6_MAXREF_READ, ID_MAXREF_WRITE := AIC_I6_MAXREF_WRITE, stObjMinRaw := NumberVariable_AIC_I06_MINRAW_N, stObjMidRaw := NumberVariable_AIC_I06_MIDRAW_N, stObjMaxRaw := NumberVariable_AIC_I06_MAXRAW_N, ID_MIN_RAW_WRITE := AIC_I6_MIN_RAW_WRITE, ID_MID_RAW_WRITE := AIC_I6_MID_RAW_WRITE, ID_MAX_RAW_WRITE := AIC_I6_MAX_RAW_WRITE);
    AnalogChannel_I7 : MyLib::sys::logiBUS_AI_Calibrate_3P_IDA_OPC(u16ObjId_RAWVAR := NumberVariable_AIC_RAW_I07, stObjCal := NumberVariable_AIC_CAL_I07_N, u16ObjId_C_MIN := Button_AIC_I07_CO, u16ObjId_C_MID := Button_AIC_I07_MID, u16ObjId_C_MAX := Button_AIC_I07_CS, Input := AnalogInput_I7, sSection := 'AI_Calibrate_3P_I7', ID_RAW_WRITE := AIC_I7_RAW_WRITE, ID_CAL_WRITE := AIC_I7_CAL_WRITE, ID_MIN_METHOD := AIC_I7_MIN_METHOD, ID_MID_TRIGGER_METHOD := AIC_I7_MID_METHOD, ID_MAX_METHOD := AIC_I7_MAX_METHOD, stObjMinRef := NumberVariable_AIC_I07_ZERO_N, stObjMidRef := NumberVariable_AIC_I07_MID_N, stObjMaxRef := NumberVariable_AIC_I07_SPAN_N, ID_MINREF_READ := AIC_I7_MINREF_READ, ID_MINREF_WRITE := AIC_I7_MINREF_WRITE, ID_MIDREF_READ := AIC_I7_MIDREF_READ, ID_MIDREF_WRITE := AIC_I7_MIDREF_WRITE, ID_MAXREF_READ := AIC_I7_MAXREF_READ, ID_MAXREF_WRITE := AIC_I7_MAXREF_WRITE, stObjMinRaw := NumberVariable_AIC_I07_MINRAW_N, stObjMidRaw := NumberVariable_AIC_I07_MIDRAW_N, stObjMaxRaw := NumberVariable_AIC_I07_MAXRAW_N, ID_MIN_RAW_WRITE := AIC_I7_MIN_RAW_WRITE, ID_MID_RAW_WRITE := AIC_I7_MID_RAW_WRITE, ID_MAX_RAW_WRITE := AIC_I7_MAX_RAW_WRITE);
    AnalogChannel_I8 : MyLib::sys::logiBUS_AI_Calibrate_3P_IDA_OPC(u16ObjId_RAWVAR := NumberVariable_AIC_RAW_I08, stObjCal := NumberVariable_AIC_CAL_I08_N, u16ObjId_C_MIN := Button_AIC_I08_CO, u16ObjId_C_MID := Button_AIC_I08_MID, u16ObjId_C_MAX := Button_AIC_I08_CS, Input := AnalogInput_I8, sSection := 'AI_Calibrate_3P_I8', ID_RAW_WRITE := AIC_I8_RAW_WRITE, ID_CAL_WRITE := AIC_I8_CAL_WRITE, ID_MIN_METHOD := AIC_I8_MIN_METHOD, ID_MID_TRIGGER_METHOD := AIC_I8_MID_METHOD, ID_MAX_METHOD := AIC_I8_MAX_METHOD, stObjMinRef := NumberVariable_AIC_I08_ZERO_N, stObjMidRef := NumberVariable_AIC_I08_MID_N, stObjMaxRef := NumberVariable_AIC_I08_SPAN_N, ID_MINREF_READ := AIC_I8_MINREF_READ, ID_MINREF_WRITE := AIC_I8_MINREF_WRITE, ID_MIDREF_READ := AIC_I8_MIDREF_READ, ID_MIDREF_WRITE := AIC_I8_MIDREF_WRITE, ID_MAXREF_READ := AIC_I8_MAXREF_READ, ID_MAXREF_WRITE := AIC_I8_MAXREF_WRITE, stObjMinRaw := NumberVariable_AIC_I08_MINRAW_N, stObjMidRaw := NumberVariable_AIC_I08_MIDRAW_N, stObjMaxRaw := NumberVariable_AIC_I08_MAXRAW_N, ID_MIN_RAW_WRITE := AIC_I8_MIN_RAW_WRITE, ID_MID_RAW_WRITE := AIC_I8_MID_RAW_WRITE, ID_MAX_RAW_WRITE := AIC_I8_MAX_RAW_WRITE);
    Output_Q1 : MyLib::sys::Button_IXA_TO_logiBUS_QXA_BG_OPC(u16ObjId := Button_Q01, Output := Output_Q1, ID_READ := Q01_READ, ID_WRITE := Q01_WRITE);
    Output_Q2 : MyLib::sys::Button_IXA_TO_logiBUS_QXA_BG_OPC(u16ObjId := Button_Q02, Output := Output_Q2, ID_READ := Q02_READ, ID_WRITE := Q02_WRITE);
    Output_Q3 : MyLib::sys::Button_IXA_TO_logiBUS_QXA_BG_OPC(u16ObjId := Button_Q03, Output := Output_Q3, ID_READ := Q03_READ, ID_WRITE := Q03_WRITE);
    Output_Q4 : MyLib::sys::Button_IXA_TO_logiBUS_QXA_BG_OPC(u16ObjId := Button_Q04, Output := Output_Q4, ID_READ := Q04_READ, ID_WRITE := Q04_WRITE);
    Output_Q5 : MyLib::sys::Button_IXA_TO_logiBUS_QXA_BG_OPC(u16ObjId := Button_Q05, Output := Output_Q5, ID_READ := Q05_READ, ID_WRITE := Q05_WRITE);
    Output_Q6 : MyLib::sys::Button_IXA_TO_logiBUS_QXA_BG_OPC(u16ObjId := Button_Q06, Output := Output_Q6, ID_READ := Q06_READ, ID_WRITE := Q06_WRITE);
    Output_Q7 : MyLib::sys::Button_IXA_TO_logiBUS_QXA_BG_OPC(u16ObjId := Button_Q07, Output := Output_Q7, ID_READ := Q07_READ, ID_WRITE := Q07_WRITE);
    Output_Q8 : MyLib::sys::Button_IXA_TO_logiBUS_QXA_BG_OPC(u16ObjId := Button_Q08, Output := Output_Q8, ID_READ := Q08_READ, ID_WRITE := Q08_WRITE);
    Output_Q9 : MyLib::sys::Button_IXA_TO_logiBUS_QXA_BG_OPC(u16ObjId := Button_Q09, Output := Output_Q9, ID_READ := Q09_READ, ID_WRITE := Q09_WRITE);
    Output_Q10 : MyLib::sys::Button_IXA_TO_logiBUS_QXA_BG_OPC(u16ObjId := Button_Q10, Output := Output_Q10, ID_READ := Q10_READ, ID_WRITE := Q10_WRITE);
    Output_Q11 : MyLib::sys::Button_IXA_TO_logiBUS_QXA_BG_OPC(u16ObjId := Button_Q11, Output := Output_Q11, ID_READ := Q11_READ, ID_WRITE := Q11_WRITE);
    Output_Q12 : MyLib::sys::Button_IXA_TO_logiBUS_QXA_BG_OPC(u16ObjId := Button_Q12, Output := Output_Q12, ID_READ := Q12_READ, ID_WRITE := Q12_WRITE);
    SystemTickSender : MyLib::sys::SystemTickSender_ISO_OPC(u16ObjId := OutputNumber_Tick, ID_WRITE := Tick_WRITE);
  END_SUBAPPS
END_SUBAPPLICATION
